// TwinCAT 3 PLC project PLC_Project
// ProgramVersion: 3.1.0.8
// libraries:
//   Tc2_MC2, * (Beckhoff Automation GmbH)
//   Tc2_Standard, * (Beckhoff Automation GmbH)
//   Tc2_System, * (Beckhoff Automation GmbH)
//   Tc3_Interfaces, * (Beckhoff Automation GmbH)
//   Tc3_Module, * (Beckhoff Automation GmbH)
// project tree:
//   DUTs/ Motion_Axis.TcDUT (not stored), Motion_AxisGroup.TcDUT (not stored), Motion_FunctionResult.TcDUT, Motion_HmiToPlc.TcDUT, Motion_PlcToHmi.TcDUT
//   GVLs/ IO_DigiIn_GVL.TcGVL, IO_DigiOut_GVL.TcGVL, Motion_GVL.TcGVL, Motion_Parameters.TcGVL
//   / PlcTask.TcTTO
//   POUs/ MAIN.TcPOU, MotionControl.TcPOU
// real-time tasks:
//   TASK PlcTask: cycle T#10ms, priority 20, ADS port 350
//   TASK OtherTask: cycle T#10ms, priority 19, ADS port 351
//   TASK PlcTask1: cycle T#4ms, priority 22, ADS port 352
//   TASK SerialTask: cycle T#2ms, priority 1, ADS port 353
// motion (NC):
//   TASK NC-Task 1 SAF: cycle T#2ms, priority 4, ADS port 501
//   TASK NC-Task 1 SVB: cycle T#10ms, priority 8, ADS port 511
//   AXIS EL7201 (id 4)
//     General: UnitName=°
//     Dynamic: Acceleration=8500, Deceleration=8500, Jerk=72250, DelayTime=0.006
//     Velo: RefSearch=360, RefSync=360, Maximum=16000
//     OtherSettings: AllowMotionCmdToSlave=true
//     encoder EncType=19
//       EncPara: ScaleFactorNumerator=360, ScaleFactorDenominator=1048576, MaxCount=#xffffffff
//     drive DrvType=16
//       DrvPara: MaxCount=#xffffffff
//         Analog: VeloReferenz=18000
//         TimeComp: TaskDelayCycles=1
//     controller CtrType=1
//       CtrPara: PriorControlFactor=1
//         PosDiffControl: Enable=false
//         Observer: BandWidth=20
//   AXIS EL7031 (id 5)
//     General: UnitName=°
//     Dynamic: Acceleration=4300, Deceleration=4300, Jerk=18490, DelayTime=0.006
//     Velo: RefSearch=360, RefSync=360, Maximum=3300
//     OtherSettings: AllowMotionCmdToSlave=true
//     encoder EncType=1
//       EncPara: ScaleFactorNumerator=1.8, ScaleFactorDenominator=64
//         Inc: RefSoftSyncMask=#x0000ffff
//     drive DrvType=5
//       Analog: VeloReferenz=3600
//       TimeComp: TaskDelayCycles=1
//     controller CtrType=1
//       CtrPara: PriorControlFactor=1
//         PosDiffControl: Enable=false
//         Observer: BandWidth=20
//   AXIS AX1 (id 1)
//     OtherSettings: AllowMotionCmdToSlave=true
//     encoder EncType=1
//     drive DrvType=5
//     controller CtrType=1
//       CtrPara: PriorControlFactor=1
//         Observer: BandWidth=20
//   AXIS AX2 (id 2)
//     OtherSettings: AllowMotionCmdToSlave=true
//     encoder EncType=1
//     drive DrvType=5
//     controller CtrType=1
//       CtrPara: PriorControlFactor=1
//         Observer: BandWidth=20
//   AXIS AX3 (id 3)
//     OtherSettings: AllowMotionCmdToSlave=true
//     encoder EncType=1
//     drive DrvType=5
//     controller CtrType=1
//       CtrPara: PriorControlFactor=1
//         Observer: BandWidth=20
//   AXIS AX4 (id 6)
//     OtherSettings: AllowMotionCmdToSlave=true
//     encoder EncType=1
//     drive DrvType=5
//     controller CtrType=1
//       CtrPara: PriorControlFactor=1
//         Observer: BandWidth=20
//   AXIS AX5 (id 7)
//     OtherSettings: AllowMotionCmdToSlave=true
//     encoder EncType=1
//     drive DrvType=5
//     controller CtrType=1
//       CtrPara: PriorControlFactor=1
//         Observer: BandWidth=20
// variable links:
//   PLC Project/PLC Project Instance <-> NC-Task 1 SAF/Axes/AX1
//     PlcTask Inputs/Motion_GVL.AXIS[1].AXIS.NcToPlc <-> Outputs/ToPlc
//     PlcTask Outputs/Motion_GVL.AXIS[1].AXIS.PlcToNc <-> Inputs/FromPlc
//   PLC Project/PLC Project Instance <-> NC-Task 1 SAF/Axes/AX2
//     PlcTask Inputs/Motion_GVL.AXIS[2].AXIS.NcToPlc <-> Outputs/ToPlc
//     PlcTask Outputs/Motion_GVL.AXIS[2].AXIS.PlcToNc <-> Inputs/FromPlc
//   PLC Project/PLC Project Instance <-> NC-Task 1 SAF/Axes/AX3
//     PlcTask Inputs/Motion_GVL.AXIS[3].AXIS.NcToPlc <-> Outputs/ToPlc
//     PlcTask Outputs/Motion_GVL.AXIS[3].AXIS.PlcToNc <-> Inputs/FromPlc
//   PLC Project/PLC Project Instance <-> NC-Task 1 SAF/Axes/AX4
//     PlcTask Inputs/Motion_GVL.AXIS[4].AXIS.NcToPlc <-> Outputs/ToPlc
//     PlcTask Outputs/Motion_GVL.AXIS[4].AXIS.PlcToNc <-> Inputs/FromPlc
//   PLC Project/PLC Project Instance <-> NC-Task 1 SAF/Axes/AX5
//     PlcTask Inputs/Motion_GVL.AXIS[5].AXIS.NcToPlc <-> Outputs/ToPlc
//     PlcTask Outputs/Motion_GVL.AXIS[5].AXIS.PlcToNc <-> Inputs/FromPlc

CONFIGURATION PLC_Project
    RESOURCE PLC ON TwinCAT3
        TASK PlcTask(INTERVAL := T#10ms, PRIORITY := 20);
        PROGRAM MAIN WITH PlcTask : MAIN;
    END_RESOURCE
END_CONFIGURATION

// ---- DUTs/Motion_FunctionResult.TcDUT
TYPE Motion_FunctionResult :
(
	MOTION_OK := -1,
	MOTION_BUSY := 0,
	MOTION_UNKNOWN_AXIS,
	MOTION_UNKNOWN_AXIS_GROUP,
	MOTION_UNKNOWN_SAME_AXIS_IN_GROUP,
	MOTION_COMMAND_ABORTED,
	MOTION_ERROR
);
END_TYPE

// ---- DUTs/Motion_HmiToPlc.TcDUT
TYPE Motion_HmiToPlc :
STRUCT
	TARGET_POSITION 	: LREAL;
	TARGET_VELOCITY 	: LREAL;
	TARGET_ACCELERATION : LREAL;
	TARGET_DECELERATION	: LREAL;
	TARGET_JERK			: LREAL;
	CONTROLLER_OVERRIDE	: LREAL;
	ON					: BOOL;
	ON_FW				: BOOL;
	ON_BW				: BOOL;
	OFF					: BOOL;
	MOVE_ABS			: BOOL;
	MOVE_REL			: BOOL;
	HALT				: BOOL;
	HOME				: BOOL;
	RESET				: BOOL;
	JOG_MODE			: BOOL := FALSE;
	JOG_FW_FAST			: BOOL;
	JOG_BW_FAST			: BOOL;
	JOG_FW_SLOW			: BOOL;
	JOG_BW_SLOW			: BOOL;
END_STRUCT
END_TYPE

// ---- DUTs/Motion_PlcToHmi.TcDUT
TYPE Motion_PlcToHmi :
STRUCT
	actPos				: LREAL;
	actVelo				: LREAL;
	setPos				: LREAL; 
	setVelo 			: LREAL; 
	controller_override : LREAL;
	ErrorID				: UDINT;
	hasError			: BOOL;
	isDisabled 			: BOOL;
	isFwDisabled 		: BOOL;
	isBwDisabled 		: BOOL;
	isCalibrated		: BOOL;
	hasJob				: BOOL;
	isNotMoving 		: BOOL;
	isPositiveDirection : BOOL;
	isNegativeDirection : BOOL;            
    isInTarget 			: BOOL;            
    isInRange 			: BOOL;            
END_STRUCT
END_TYPE

// ---- GVLs/IO_DigiIn_GVL.TcGVL
VAR_GLOBAL
	Digital_Input AT %I* : ARRAY [1..10] OF BOOL;
END_VAR

// ---- GVLs/IO_DigiOut_GVL.TcGVL
VAR_GLOBAL
	Digital_Output AT %Q* : ARRAY [1..100] OF BOOL;
END_VAR

// ---- GVLs/Motion_GVL.TcGVL
VAR_GLOBAL
	HmiToPlc	: ARRAY[1..MAX_AXES] OF Motion_HmiToPlc;
	PlcToHmi	: ARRAY[1..MAX_AXES] OF Motion_PlcToHmi;
	AXIS		: ARRAY[1..MAX_AXES] OF Motion_Axis;
END_VAR

// ---- GVLs/Motion_Parameters.TcGVL
VAR_GLOBAL CONSTANT
	MAX_AXES 		: INT := 5;
	MAX_AXIS_GROUPS	: INT := 1;
END_VAR

// ---- POUs/MAIN.TcPOU
PROGRAM MAIN
VAR
	basgMotion : MotionControl;
	i: INT;
END_VAR

basgMotion(HMI_MODE:=TRUE);

END_PROGRAM

// ---- POUs/MotionControl.TcPOU
FUNCTION_BLOCK MotionControl
VAR_INPUT
	HMI_MODE : BOOL;
END_VAR
VAR_OUTPUT
END_VAR
VAR
	fbPower 	: ARRAY [1..MAX_AXES] OF MC_POWER;
	fbReset 	: ARRAY [1..MAX_AXES] OF MC_RESET;
	fbHome		: ARRAY	[1..MAX_AXES] OF MC_HOME;
	fbMoveA 	: ARRAY [1..MAX_AXES] OF MC_MOVEABSOLUTE;
	fbMoveR 	: ARRAY [1..MAX_AXES] OF MC_MOVERELATIVE;
	fbJog		: ARRAY [1..MAX_AXES] OF MC_JOG;
	fbHalt	 	: ARRAY [1..MAX_AXES] OF MC_HALT;
	i			: INT;
END_VAR

IF HMI_MODE THEN 
	FOR i := 1 TO MAX_AXES BY 1 DO
		ACT_UpdateStatus();
		IF HmiToPlc[i].OFF THEN
			ACT_Off();
		ELSIF HmiToPlc[i].ON THEN 
			ACT_On();
		END_IF
		IF NOT HmiToPlc[i].JOG_MODE THEN 
			Jog_Stop(i);
			IF HmiToPlc[i].HALT THEN 
				ACT_Halt();
			ELSIF HmiToPlc[i].MOVE_ABS THEN
				ACT_MoveToPosition();
			END_IF
			IF HmiToPlc[i].MOVE_REL THEN
				ACT_MoveByDistance();
			END_IF
		ELSE
			ACT_Jog();
		END_IF
	END_FOR
END_IF

ACTION ACT_MoveByDistance:
CASE MoveByDistance(i,HmiToPlc[i].TARGET_POSITION,HmiToPlc[i].TARGET_VELOCITY,HmiToPlc[i].TARGET_ACCELERATION,HmiToPlc[i].TARGET_DECELERATION,HmiToPlc[i].TARGET_JERK) OF
Motion_FunctionResult.MOTION_UNKNOWN_AXIS:
	HmiToPlc[i].MOVE_REL := FALSE;
Motion_FunctionResult.MOTION_COMMAND_ABORTED: 
	HmiToPlc[i].MOVE_REL := FALSE;
Motion_FunctionResult.MOTION_ERROR:
	HmiToPlc[i].MOVE_REL := FALSE;
Motion_FunctionResult.MOTION_BUSY: 
	;
Motion_FunctionResult.MOTION_OK:
	HmiToPlc[i].MOVE_REL := FALSE;
END_CASE
END_ACTION

METHOD PUBLIC MoveToPosition : Motion_FunctionResult
VAR_INPUT
	INDEX 			: INT;
	POSITION		: LREAL;
	VELOCITY		: LREAL;
	ACCELERATION	: LREAL;
	DECELERATION	: LREAL;
	JERK			: LREAL;
END_VAR
IF INDEX > MAX_AXES OR INDEX < 1 AND VELOCITY <= 0 THEN 
	MoveToPosition := Motion_FunctionResult.MOTION_UNKNOWN_AXIS;
ELSE
	fbMoveA[INDEX](
		Axis:= AXIS[INDEX].AXIS, 
		Execute:= TRUE, 
		Position:= POSITION, 
		Velocity:= VELOCITY, 
		Acceleration:= ACCELERATION, 
		Deceleration:= DECELERATION, 
		Jerk:= JERK );
	IF fbMoveA[INDEX].Error THEN
		fbMoveA[INDEX](
			Axis:= AXIS[INDEX].AXIS, 
			Execute:= FALSE );
		MoveToPosition := Motion_FunctionResult.MOTION_ERROR;
	ELSIF fbMoveA[INDEX].CommandAborted THEN
		fbMoveA[INDEX](
			Axis:= AXIS[INDEX].AXIS, 
			Execute:= FALSE );
		MoveToPosition := Motion_FunctionResult.MOTION_COMMAND_ABORTED;
	ELSIF fbMoveA[INDEX].Done THEN
		fbMoveA[INDEX](
			Axis:= AXIS[INDEX].AXIS, 
			Execute:= FALSE );
		MoveToPosition := Motion_FunctionResult.MOTION_OK;
	ELSE
		MoveToPosition := Motion_FunctionResult.MOTION_BUSY;
	END_IF
END_IF
END_METHOD

ACTION ACT_On:
On(i, HmiToPlc[i].ON_FW, HmiToPlc[i].ON_BW, HmiToPlc[i].CONTROLLER_OVERRIDE);
END_ACTION

METHOD PUBLIC Jog_Stop : Motion_FunctionResult
VAR_INPUT
	INDEX : INT;
END_VAR
fbJog[INDEX](
	Axis:= AXIS[INDEX].AXIS, 
	JogForward:= FALSE, 
	JogBackwards:= FALSE );
IF fbJog[INDEX].Error THEN 
	Jog_Stop := Motion_FunctionResult.MOTION_ERROR;
ELSE
	Jog_Stop := Motion_FunctionResult.MOTION_OK;
END_IF
END_METHOD

METHOD PUBLIC Home : Motion_FunctionResult
VAR_INPUT
	INDEX : INT;
END_VAR
IF INDEX > MAX_AXES OR INDEX < 1 THEN 
	Home := Motion_FunctionResult.MOTION_UNKNOWN_AXIS;
ELSE
	fbHome[INDEX](
		Axis:= AXIS[INDEX].AXIS, 
		Execute:= TRUE, 
		Position:= 0, 
		HomingMode:= MC_DefaultHoming, 
		bCalibrationCam:= AXIS[INDEX].HOME_CALIBRATION );
	IF fbHome[INDEX].Error THEN
		fbHome[INDEX](
			Axis:= AXIS[INDEX].AXIS, 
			Execute:= FALSE );
		Home := Motion_FunctionResult.MOTION_ERROR;
	ELSIF fbHome[INDEX].CommandAborted THEN
		fbHome[INDEX](
			Axis:= AXIS[INDEX].AXIS, 
			Execute:= FALSE );
		Home := Motion_FunctionResult.MOTION_COMMAND_ABORTED;
	ELSIF fbHome[INDEX].Done THEN
		fbHome[INDEX](
			Axis:= AXIS[INDEX].AXIS, 
			Execute:= FALSE );
		Home := Motion_FunctionResult.MOTION_OK;
	ELSE
		Home := Motion_FunctionResult.MOTION_BUSY;
	END_IF
END_IF
END_METHOD

ACTION ACT_Halt:
CASE Halt(i) OF 
Motion_FunctionResult.MOTION_UNKNOWN_AXIS:
	HmiToPlc[i].HALT := FALSE;
Motion_FunctionResult.MOTION_ERROR:
	HmiToPlc[i].HALT := FALSE;
Motion_FunctionResult.MOTION_OK:
	HmiToPlc[i].HALT := FALSE;
Motion_FunctionResult.MOTION_COMMAND_ABORTED:
	HmiToPlc[i].HALT := FALSE;
Motion_FunctionResult.MOTION_BUSY:
	;
END_CASE
HmiToPlc[i].MOVE_ABS := FALSE;
HmiToPlc[i].MOVE_REL := FALSE;
END_ACTION

PROPERTY AxisGroup_Count : INT
GET
AXISGROUP_Count := MAX_AXIS_GROUPS;
END_GET
END_PROPERTY

ACTION ACT_Off:
Off(i);
END_ACTION

ACTION ACT_MoveToPosition:
CASE MoveToPosition(i,HmiToPlc[i].TARGET_POSITION,HmiToPlc[i].TARGET_VELOCITY,HmiToPlc[i].TARGET_ACCELERATION,HmiToPlc[i].TARGET_DECELERATION,HmiToPlc[i].TARGET_JERK) OF
Motion_FunctionResult.MOTION_UNKNOWN_AXIS:
	HmiToPlc[i].MOVE_ABS := FALSE;
Motion_FunctionResult.MOTION_COMMAND_ABORTED: 
	HmiToPlc[i].MOVE_ABS := FALSE;
Motion_FunctionResult.MOTION_ERROR:
	HmiToPlc[i].MOVE_ABS := FALSE;
Motion_FunctionResult.MOTION_BUSY: 
	;
Motion_FunctionResult.MOTION_OK:
	HmiToPlc[i].MOVE_ABS := FALSE;
END_CASE
END_ACTION

ACTION ACT_Reset:
IF Reset(i) = Motion_FunctionResult.MOTION_OK THEN
	HmiToPlc[i].RESET := FALSE;
END_IF
END_ACTION

PROPERTY PUBLIC AXIS_COUNT : INT
GET
AXIS_COUNT := MAX_AXES;
END_GET
END_PROPERTY

ACTION ACT_UpdateStatus:
AXIS[i].AXIS.ReadStatus();
PlcToHmi[i].actPos	:= AXIS[i].AXIS.NcToPlc.ActPos;
PlcToHmi[i].actVelo := AXIS[i].AXIS.NcToPlc.ActVelo;
PlcToHmi[i].setPos	:= AXIS[i].AXIS.NcToPlc.SetPos;
PlcToHmi[i].setVelo := AXIS[i].AXIS.NcToPlc.SetVelo;
PlcToHmi[i].controller_override := fbPower[i].Override;
PlcToHmi[i].hasError := AXIS[i].AXIS.Status.Error;
PlcToHmi[i].ErrorID := AXIS[i].AXIS.Status.ErrorID;
PlcToHmi[i].isBwDisabled := NOT fbPower[i].Enable_Negative;
PlcToHmi[i].isFwDisabled := NOT fbPower[i].Enable_Positive;
PlcToHmi[i].isCalibrated := AXIS[i].AXIS.Status.Homed;
PlcToHmi[i].isDisabled := AXIS[i].AXIS.Status.Disabled;
PlcToHmi[i].isInRange := AXIS[i].AXIS.Status.InPositionArea;
PlcToHmi[i].isInTarget := AXIS[i].AXIS.Status.InTargetPosition;
PlcToHmi[i].isNegativeDirection := AXIS[i].AXIS.Status.NegativeDirection;
PlcToHmi[i].isNotMoving := AXIS[i].AXIS.Status.NotMoving;
PlcToHmi[i].isPositiveDirection := AXIS[i].AXIS.Status.PositiveDirection;
END_ACTION

METHOD On : Motion_FunctionResult
VAR_INPUT
	INDEX : INT;
	ENABLE_FW 	: BOOL;
	ENABLE_BW	: BOOL;
	OVERRIDE	: LREAL;
END_VAR
IF INDEX > MAX_AXES OR INDEX < 1 THEN 
	On := Motion_FunctionResult.MOTION_UNKNOWN_AXIS;
ELSE
	fbPower[INDEX](
		Axis:= AXIS[INDEX].AXIS, 
		Enable:= TRUE, 
		Enable_Positive:= ENABLE_FW, 
		Enable_Negative:= ENABLE_BW, 
		Override:= OVERRIDE );
	IF fbPower[INDEX].Error THEN
		On := Motion_FunctionResult.MOTION_ERROR;
	ELSIF fbPower[INDEX].Status THEN
		On := Motion_FunctionResult.MOTION_OK;
	ELSE
		On := Motion_FunctionResult.MOTION_BUSY;
	END_IF
END_IF
END_METHOD

ACTION ACT_Jog:
IF HmiToPlc[i].JOG_FW_FAST THEN
	Jog_Start(i, FALSE, TRUE);
ELSIF HmiToPlc[i].JOG_FW_SLOW THEN
	Jog_Start(i, FALSE, FALSE);
ELSIF HmiToPlc[i].JOG_BW_FAST THEN
	Jog_Start(i, TRUE, TRUE);
ELSIF HmiToPlc[i].JOG_BW_SLOW THEN
	Jog_Start(i, TRUE, FALSE);
ELSE
	Jog_Stop(i);
END_IF
END_ACTION

METHOD PUBLIC Reset : Motion_FunctionResult
VAR_INPUT
	INDEX :INT;
END_VAR
IF INDEX > MAX_AXES OR INDEX < 1 THEN 
	Reset := Motion_FunctionResult.MOTION_UNKNOWN_AXIS;
ELSE
	fbReset[INDEX](
		Axis:= AXIS[INDEX].AXIS, 
		Execute:= TRUE );
	IF fbReset[INDEX].Error THEN
		fbReset[INDEX](
			Axis:= AXIS[INDEX].AXIS, 
			Execute:= FALSE );
		Reset := Motion_FunctionResult.MOTION_ERROR;
	ELSIF fbReset[INDEX].Done THEN
		fbReset[INDEX](
			Axis:= AXIS[INDEX].AXIS, 
			Execute:= FALSE );
		Reset := Motion_FunctionResult.MOTION_OK;
	ELSE
		Reset := Motion_FunctionResult.MOTION_BUSY;
	END_IF
END_IF
END_METHOD

METHOD PUBLIC Halt : Motion_FunctionResult
VAR_INPUT
	INDEX : INT;
END_VAR
IF INDEX > MAX_AXES OR INDEX < 1 THEN 
	Halt := Motion_FunctionResult.MOTION_UNKNOWN_AXIS;
ELSE
	fbHalt[INDEX](
		Axis:= AXIS[INDEX].AXIS, 
		Execute:= TRUE );
	fbMoveA[INDEX](
		Axis:= AXIS[INDEX].AXIS, 
		Execute:= FALSE );
	fbMoveR[INDEX](
		Axis:= AXIS[INDEX].AXIS, 
		Execute:= FALSE );
	IF fbHalt[INDEX].Error THEN
		fbHalt[INDEX](
			Axis:= AXIS[INDEX].AXIS, 
			Execute:= FALSE );
		Halt := Motion_FunctionResult.MOTION_ERROR;
	ELSIF fbHalt[INDEX].CommandAborted THEN
		fbHalt[INDEX](
			Axis:= AXIS[INDEX].AXIS, 
			Execute:= FALSE );
		Halt := Motion_FunctionResult.MOTION_COMMAND_ABORTED;
	ELSIF fbHalt[INDEX].Done THEN
		fbHalt[INDEX](
			Axis:= AXIS[INDEX].AXIS, 
			Execute:= FALSE );
		Halt := Motion_FunctionResult.MOTION_OK;
	ELSE
		Halt := Motion_FunctionResult.MOTION_BUSY;
	END_IF
END_IF
END_METHOD

METHOD PUBLIC MoveByDistance : Motion_FunctionResult
VAR_INPUT
	INDEX 			: INT;
	DISTANCE 		: LREAL;
	VELOCITY 		: LREAL;
	ACCELERATION 	: LREAL;
	DECELERATION 	: LREAL;
	JERK 			: LREAL;
END_VAR
IF INDEX > MAX_AXES OR INDEX < 1 AND VELOCITY <= 0 THEN 
	MoveByDistance := Motion_FunctionResult.MOTION_UNKNOWN_AXIS;
ELSE
	fbMoveR[INDEX](
		Axis:= AXIS[INDEX].AXIS, 
		Execute:= TRUE, 
		Distance:= DISTANCE, 
		Velocity:= VELOCITY, 
		Acceleration:= ACCELERATION, 
		Deceleration:= DECELERATION, 
		Jerk:= JERK );
	IF fbMoveR[INDEX].Error THEN
		fbMoveR[INDEX](
			Axis:= AXIS[INDEX].AXIS, 
			Execute:= FALSE );
		MoveByDistance := Motion_FunctionResult.MOTION_ERROR;
	ELSIF fbMoveR[INDEX].CommandAborted THEN
		fbMoveR[INDEX](
			Axis:= AXIS[INDEX].AXIS, 
			Execute:= FALSE );
		MoveByDistance := Motion_FunctionResult.MOTION_COMMAND_ABORTED;
	ELSIF fbMoveR[INDEX].Done THEN
		fbMoveR[INDEX](
			Axis:= AXIS[INDEX].AXIS, 
			Execute:= FALSE );
		MoveByDistance := Motion_FunctionResult.MOTION_OK;
	ELSE
		MoveByDistance := Motion_FunctionResult.MOTION_BUSY;
	END_IF
END_IF
END_METHOD

METHOD PUBLIC Off : Motion_FunctionResult
VAR_INPUT
	INDEX : INT;
END_VAR
IF INDEX > MAX_AXES OR INDEX < 1 THEN 
	Off := Motion_FunctionResult.MOTION_UNKNOWN_AXIS;
ELSE
	fbPower[INDEX](
		Axis:= AXIS[INDEX].AXIS, 
		Enable:= FALSE, 
		Enable_Positive:= FALSE, 
		Enable_Negative:= FALSE, 
		Override:= 0 );
	IF fbPower[INDEX].Error THEN
		Off := Motion_FunctionResult.MOTION_ERROR;
	ELSIF NOT fbPower[INDEX].Status THEN
		Off := Motion_FunctionResult.MOTION_OK;
	ELSE
		Off := Motion_FunctionResult.MOTION_BUSY;
	END_IF
END_IF
END_METHOD

METHOD PUBLIC Jog_Start : Motion_FunctionResult
VAR_INPUT
	INDEX		: INT;
	REVERSE		: BOOL := FALSE;
	FAST_MODE	: BOOL := FALSE;
END_VAR
IF FAST_MODE THEN 
	fbJog[INDEX].Mode := MC_JOGMODE_STANDARD_FAST;
ELSE
	fbJog[INDEX].Mode := MC_JOGMODE_STANDARD_SLOW;
END_IF

fbJog[INDEX](
	Axis:= AXIS[INDEX].AXIS, 
	JogForward:= NOT REVERSE, 
	JogBackwards:= REVERSE );
IF fbJog[INDEX].Error THEN 
	Jog_Start := Motion_FunctionResult.MOTION_ERROR;
ELSIF AXIS[INDEX].AXIS.Status.Moving THEN 
	Jog_Start := Motion_FunctionResult.MOTION_OK;
END_IF
END_METHOD

END_FUNCTION_BLOCK
